KUKA KRL program: exampleKukaPath.src, exampleKukaPath.dat

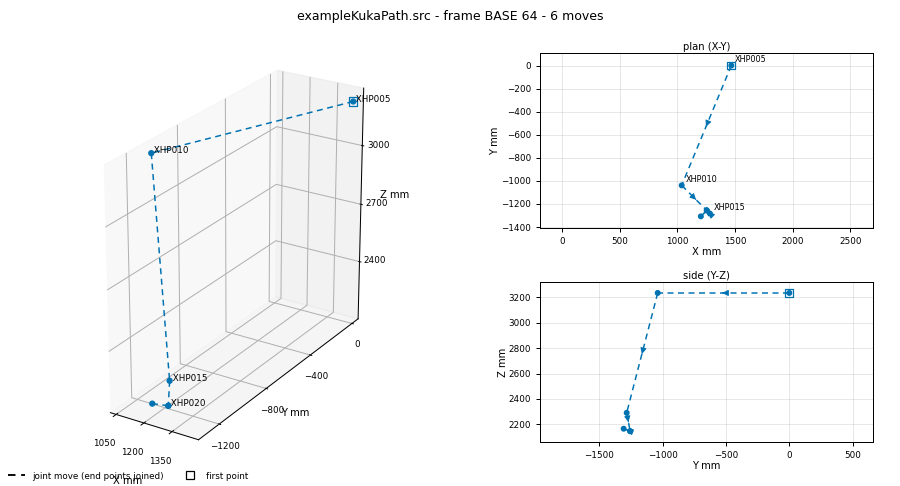
[picture p0: tool path of exampleKukaPath.src in frame BASE 64, 6 of 6 moves have a stored position in this frame; points joined in program order, loops and branches not executed]
--- exampleKukaPath.src ---
&ACCESS RVO1
&REL 274
&COMMENT Bld
&PARAM DISKPATH = KRC:\R1\Program\Production\223
DEF msn223v_030_01_030r2( )

DECL INT SRCDATA
DECL FLOAT SCRDATAFLOAT, ADRa
DECL INT DATAS13

;FOLD INI
  ;FOLD BASISTECH INI
    GLOBAL INTERRUPT DECL 3 WHEN $IN[1]==TRUE DO IR_STOPM ( )
    INTERRUPT ON 3
    BAS (#INITMOV,0 )
  ;ENDFOLD (BASISTECH INI)
  ;FOLD USER INI
    ;Make your modifications here
  ;ENDFOLD (USER INI)
;ENDFOLD (INI)

WAIT FOR  ( $IN[126] )
$OUT[125]=TRUE
$OUT[161]=FALSE

COLLSTOP( 15, 1 ) ;not Interrupt-Controlled
USE_CD_PARAMS(1)

;FOLD PTP HP005 CONT Vel=100 % PDATHH Tool[64]:NULL [64]:NULL ;%{PE}
;FOLD Parameters ;%{h}
;Params IlfProvider=kukaroboter.basistech.inlineforms.movement.old; Kuka.IsGlobalPoint=False; Kuka.PointName=HP005; Kuka.BlendingEnabled=True; Kuka.MoveDataPtpName=PDATHH; Kuka.VelocityPtp=100; Kuka.CurrentCDSetIndex=0; Kuka.MovementParameterFieldEnabled=True; IlfCommand=PTP
;ENDFOLD
$BWDSTART = FALSE
PDAT_ACT = PPDATHH
FDAT_ACT = FHP005
BAS(#PTP_PARAMS, 100.0)
SET_CD_PARAMS (0)
PTP XHP005 C_DIS C_DIS
;ENDFOLD

;FOLD PTP HP010 CONT Vel=100 % PDATHH Tool[64]:NULL Base[64]:NULL ;%{PE}
;FOLD Parameters ;%{h}
;Params IlfProvider=kukaroboter.basistech.inlineforms.movement.old; Kuka.IsGlobalPoint=False; Kuka.PointName=HP010; Kuka.BlendingEnabled=True; Kuka.MoveDataPtpName=PDATHH; Kuka.VelocityPtp=100; Kuka.CurrentCDSetIndex=0; Kuka.MovementParameterFieldEnabled=True; IlfCommand=PTP
;ENDFOLD
$BWDSTART = FALSE
PDAT_ACT = PPDATHH
FDAT_ACT = FHP010
BAS(#PTP_PARAMS, 100.0)
SET_CD_PARAMS (0)
PTP XHP010 C_Dis
;ENDFOLD
;FOLD PTP HP015 CONT Vel=100 % PDATHH Tool[64]:NULL Base[64]: ;%{PE}
;FOLD Parameters ;%{h}
;Params IlfProvider=kukaroboter.basistech.inlineforms.movement.old; Kuka.IsGlobalPoint=False; Kuka.PointName=HP015; Kuka.BlendingEnabled=True; Kuka.MoveDataPtpName=PDATHH; Kuka.VelocityPtp=100; Kuka.CurrentCDSetIndex=0; Kuka.MovementParameterFieldEnabled=True; IlfCommand=PTP
;ENDFOLD
$BWDSTART = FALSE
PDAT_ACT = PPDATHH
FDAT_ACT = FHP015
BAS(#PTP_PARAMS, 100.0)
SET_CD_PARAMS (0)
PTP XHP015 C_Dis
;ENDFOLD
;FOLD PTP HP020 CONT Vel=100 % PDATHH Tool[64]:NULL Base[64]: ;%{PE}
;FOLD Parameters ;%{h}
;Params IlfProvider=kukaroboter.basistech.inlineforms.movement.old; Kuka.IsGlobalPoint=False; Kuka.PointName=HP020; Kuka.BlendingEnabled=True; Kuka.MoveDataPtpName=PDATHH; Kuka.VelocityPtp=100; Kuka.CurrentCDSetIndex=0; Kuka.MovementParameterFieldEnabled=True; IlfCommand=PTP
;ENDFOLD
$BWDSTART = FALSE
PDAT_ACT = PPDATHH
FDAT_ACT = FHP020
BAS(#PTP_PARAMS, 100.0)
SET_CD_PARAMS (0)
PTP XHP020 C_Dis
;ENDFOLD
;FOLD PTP HP025 Vel=100 % PDATHH Tool[64]:NULL Base[64]: ;%{PE}
;FOLD Parameters ;%{h}
;Params IlfProvider=kukaroboter.basistech.inlineforms.movement.old; Kuka.IsGlobalPoint=False; Kuka.PointName=HP025; Kuka.BlendingEnabled=False; Kuka.MoveDataPtpName=PDATHH; Kuka.VelocityPtp=100; Kuka.CurrentCDSetIndex=0; Kuka.MovementParameterFieldEnabled=True; IlfCommand=PTP
;ENDFOLD
$BWDSTART = FALSE
PDAT_ACT = PPDATHH
FDAT_ACT = FHP025
BAS(#PTP_PARAMS, 100.0)
SET_CD_PARAMS (0)
PTP XHP025
;ENDFOLD
;FOLD PTP HP030 Vel=100 % PDATHH Tool[64]:NULL Base[64]: ;%{PE}
;FOLD Parameters ;%{h}
;Params IlfProvider=kukaroboter.basistech.inlineforms.movement.old; Kuka.IsGlobalPoint=False; Kuka.PointName=HP030; Kuka.BlendingEnabled=False; Kuka.MoveDataPtpName=PDATHH; Kuka.VelocityPtp=100; Kuka.CurrentCDSetIndex=0; Kuka.MovementParameterFieldEnabled=True; IlfCommand=PTP
;ENDFOLD
$BWDSTART = FALSE
PDAT_ACT = PPDATHH
FDAT_ACT = FHP030
BAS(#PTP_PARAMS, 100.0)
SET_CD_PARAMS (0)
PTP XHP030
;ENDFOLD

$OUT[125]=TRUE
$OUT[161]=TRUE
COLLSTOP( 15, 2+0 )
USE_CD_PARAMS( 0)

END

GLOBAL DEFFCT BOOL nearE6Pos(ePOS:IN)
 DECL E6POS ePOS

 DECL E6POS Delta
 DECL BOOL bRet

 bRet = False

 Delta.X = ABS(ePOS.X - $Pos_Act.X)
 Delta.Y = ABS(ePOS.Y - $Pos_Act.Y)
 Delta.Z = ABS(ePOS.Z - $Pos_Act.Z)
 Delta.A = ABS(ePOS.A - $Pos_Act.A)
 Delta.B = ABS(ePOS.B - $Pos_Act.B)
 Delta.C = ABS(ePOS.C - $Pos_Act.C)

 Delta.S = ePOS.S - $Pos_Act.S
 Delta.T = ePOS.T - $Pos_Act.T

 Delta.E1 = ABS(ePOS.E1 - $Pos_Act.E1)
 Delta.E2 = ABS(ePOS.E2 - $Pos_Act.E2)
 Delta.E3 = ABS(ePOS.E3 - $Pos_Act.E3)
 Delta.E4 = ABS(ePOS.E4 - $Pos_Act.E4)
 Delta.E5 = ABS(ePOS.E5 - $Pos_Act.E5)
 Delta.E6 = ABS(ePOS.E6 - $Pos_Act.E6)

 bRet= (Delta.X < MaxPosTol.X) and (Delta.Y < MaxPosTol.Y) and (Delta.Z < MaxPosTol.Z) and (Delta.A < MaxPosTol.A) and (Delta.B < MaxPosTol.B) and (Delta.C < MaxPosTol.C)
 bRet=bRet and (Delta.S == 0) and (Delta.T == 0)
 bRet=bRet and (Delta.E1 < MaxPosTol.E1) and (Delta.E2 < MaxPosTol.E2) and (Delta.E3 < MaxPosTol.E3) and (Delta.E4 < MaxPosTol.E4) and (Delta.E5 < MaxPosTol.E5) and (Delta.E6 < MaxPosTol.E6)
 Return(bRet)
ENDFCT

--- exampleKukaPath.dat ---
&ACCESS RVO1
&REL 274
&COMMENT Blindnietmutter setzen
&PARAM DISKPATH = KRC:\R1\Program\Production\223
DEFDAT  MSN223V_030_01_030R2
;FOLD EXTERNAL DECLARATIONS;%{PE}%MKUKATPBASIS,%CEXT,%VCOMMON,%P

;FOLD BASISTECH EXT;%{PE}%MKUKATPBASIS,%CEXT,%VEXT,%P
EXT  BAS (BAS_COMMAND  :IN,REAL  :IN )
DECL INT SUCCESS, FAIL, PROG
;ENDFOLD (BASISTECH EXT)

;FOLD USER EXT;%{E}%MKUKATPUSER,%CEXT,%VEXT,%P
;Make here your modifications
BOOL PROC_OK=FALSE

;FOLD COLLISION
EXT  COLLSTOP (INT  :IN,INT  :IN )
;ENDFOLD  (Collision)
;ENDFOLD (USER EXT)
;ENDFOLD (EXTERNAL DECLERATIONS)

DECL BOOL $BWDSTART = FALSE
DECL PDAT PDAT_ACT ={VEL 50.0000,ACC 50.0000,APO_DIST 100.000,APO_MODE #CDIS,GEAR_JERK 100.000,EXAX_IGN 0}
DECL FDAT FDAT_ACT = {TOOL_NO 64,BASE_NO 64,IPO_FRAME #BASE,POINT2[] " "}


; E6POS declarations
DECL E6POS XHP005={X 1468.736,Y 0.0,Z 3235.954,A 0.0,B 45.0,C 0.0,S 18,T 2,E1 0.0,E2 0.0,E3 0.0,E4 0.0,E5 0.0,E6 0.0}
DECL E6POS XHP010={X 1038.553,Y -1038.553,Z 3235.954,A -45.0,B 45.0,C 0.0,S 18,T 2,E1 0.0,E2 0.0,E3 0.0,E4 0.0,E5 0.0,E6 0.0}
DECL E6POS XHP015={X 1283.399,Y -1283.399,Z 2290.000,A 0.0,B 90.0,C 45.0,S 18,T 2,E1 0.0,E2 0.0,E3 0.0,E4 0.0,E5 0.0,E6 0.0}
DECL E6POS XHP020={X 1255.926,Y -1255.926,Z 2145.000,A -45.000,B 120.000,C 0.0,S 18,T 2,E1 0.0,E2 0.0,E3 0.0,E4 0.0,E5 0.0,E6 0.0}
DECL E6POS XHP025={X 1255.926,Y -1255.926,Z 2145.000,A 4.107,B 131.410,C 40.893,S 18,T 2,E1 0.0,E2 0.0,E3 0.0,E4 0.0,E5 0.0,E6 0.0}
DECL E6POS XHP030={X 1204.661,Y -1307.191,Z 2164.426,A 16.813,B 156.452,C 61.813,S 18,T 2,E1 0.0,E2 0.0,E3 0.0,E4 0.0,E5 0.0,E6 0.0}


; FDAT declarations
DECL FDAT FHP005={TOOL_NO 64,BASE_NO 64,IPO_FRAME #BASE,POINT2[] " "}
DECL FDAT FHP010={TOOL_NO 64,BASE_NO 64,IPO_FRAME #BASE,POINT2[] " "}
DECL FDAT FHP015={TOOL_NO 64,BASE_NO 64,IPO_FRAME #BASE,POINT2[] " "}
DECL FDAT FHP020={TOOL_NO 64,BASE_NO 64,IPO_FRAME #BASE,POINT2[] " "}
DECL FDAT FHP025={TOOL_NO 64,BASE_NO 64,IPO_FRAME #BASE,POINT2[] " "}
DECL FDAT FHP030={TOOL_NO 64,BASE_NO 64,IPO_FRAME #BASE,POINT2[] " "}


; LDAT declarations
DECL LDAT LLDATHH={VEL 0.200000,ACC 100.000,APO_DIST 500.000,APO_FAC 50.0000,AXIS_VEL 100.000,AXIS_ACC 100.000,ORI_TYP #VAR,CIRC_TYP #BASE,JERK_FAC 50.0000,GEAR_JERK 100.000,EXAX_IGN 0}
DECL LDAT LLDATHM={VEL 2.00000,ACC 100.000,APO_DIST 100.000,APO_FAC 50.0000,AXIS_VEL 100.000,AXIS_ACC 100.000,ORI_TYP #VAR,CIRC_TYP #BASE,JERK_FAC 50.0000,GEAR_JERK 100.000,EXAX_IGN 0}
DECL LDAT LLDATHL={VEL 2.00000,ACC 100.000,APO_DIST 30.0000,APO_FAC 50.0000,AXIS_VEL 100.000,AXIS_ACC 100.000,ORI_TYP #VAR,CIRC_TYP #BASE,JERK_FAC 50.0000,GEAR_JERK 100.000,EXAX_IGN 0}
DECL LDAT LLDATMH={VEL 2.00000,ACC 50.0000,APO_DIST 500.000,APO_FAC 50.0000,AXIS_VEL 100.000,AXIS_ACC 100.000,ORI_TYP #VAR,CIRC_TYP #BASE,JERK_FAC 50.0000,GEAR_JERK 100.000,EXAX_IGN 0}
DECL LDAT LLDATMM={VEL 2.00000,ACC 50.0000,APO_DIST 100.000,APO_FAC 50.0000,AXIS_VEL 100.000,AXIS_ACC 100.000,ORI_TYP #VAR,CIRC_TYP #BASE,JERK_FAC 50.0000,GEAR_JERK 100.000,EXAX_IGN 0}
DECL LDAT LLDATML={VEL 2.00000,ACC 50.0000,APO_DIST 30.0000,APO_FAC 50.0000,AXIS_VEL 100.000,AXIS_ACC 100.000,ORI_TYP #VAR,CIRC_TYP #BASE,JERK_FAC 50.0000,GEAR_JERK 100.000,EXAX_IGN 0}
DECL LDAT LLDATLH={VEL 2.00000,ACC 25.0000,APO_DIST 500.000,APO_FAC 50.0000,AXIS_VEL 100.000,AXIS_ACC 100.000,ORI_TYP #VAR,CIRC_TYP #BASE,JERK_FAC 50.0000,GEAR_JERK 100.000,EXAX_IGN 0}
DECL LDAT LLDATLM={VEL 2.00000,ACC 25.0000,APO_DIST 100.000,APO_FAC 50.0000,AXIS_VEL 100.000,AXIS_ACC 100.000,ORI_TYP #VAR,CIRC_TYP #BASE,JERK_FAC 50.0000,GEAR_JERK 100.000,EXAX_IGN 0}
DECL LDAT LLDATLL={VEL 2.00000,ACC 25.0000,APO_DIST 30.0000,APO_FAC 50.0000,AXIS_VEL 100.000,AXIS_ACC 100.000,ORI_TYP #VAR,CIRC_TYP #BASE,JERK_FAC 50.0000,GEAR_JERK 100.000,EXAX_IGN 0}

; PDAT declarations
DECL PDAT PPDATHH={VEL 50.0000,ACC 50.0000,APO_DIST 100.000,APO_MODE #CDIS,GEAR_JERK 100.000,EXAX_IGN 0}
DECL PDAT PPDATHM={VEL 100.000,ACC 100.000,APO_DIST 500.000,APO_MODE #CDIS,GEAR_JERK 100.000,EXAX_IGN 0}
DECL PDAT PPDATHL={VEL 100.000,ACC 100.000,APO_DIST 100.000,APO_MODE #CDIS,GEAR_JERK 100.000,EXAX_IGN 0}
DECL PDAT PPDATMH={VEL 100.000,ACC 50.0000,APO_DIST 1000.00,APO_MODE #CDIS,GEAR_JERK 100.000,EXAX_IGN 0}
DECL PDAT PPDATMM={VEL 100.000,ACC 50.0000,APO_DIST 500.000,APO_MODE #CDIS,GEAR_JERK 100.000,EXAX_IGN 0}
DECL PDAT PPDATML={VEL 100.000,ACC 50.0000,APO_DIST 100.000,APO_MODE #CDIS,GEAR_JERK 100.000,EXAX_IGN 0}
DECL PDAT PPDATLH={VEL 100.000,ACC 25.0000,APO_DIST 1000.00,APO_MODE #CDIS,GEAR_JERK 100.000,EXAX_IGN 0}
DECL PDAT PPDATLM={VEL 100.000,ACC 25.0000,APO_DIST 500.000,APO_MODE #CDIS,GEAR_JERK 100.000,EXAX_IGN 0}
DECL PDAT PPDATLL={VEL 100.000,ACC 25.0000,APO_DIST 100.000,APO_MODE #CDIS,GEAR_JERK 100.000,EXAX_IGN 0}

DECL MODULEPARAM_T LAST_TP_PARAMS={PARAMS[] "Kuka.PointName=HP115; Kuka.FrameData.base_no=1; Kuka.FrameData.tool_no=1; Kuka.FrameData.ipo_frame=#BASE; Kuka.FrameData.point2=; Kuka.isglobalpoint=False; Kuka.MoveDataPtpName=PDATHH; Kuka.MovementDataPdat.apo_mode=#CDIS; Kuka.MovementDataPdat.apo_dist=100; Kuka.MovementData.vel=50; Kuka.MovementData.acc=50; Kuka.MovementData.gear_jerk=100; Kuka.MovementData.exax_ign=0; Kuka.VelocityPtp=50; Kuka.BlendingEnabled=False; Kuka.CurrentCDSetIndex=0; Kuka.MoveDataName=LDATHH; Kuka.MovementData.apo_fac=50; Kuka.MovementData.apo_dist=500; Kuka.MovementData.axis_acc=100; Kuka.MovementData.axis_vel=100; Kuka.MovementData.circ_typ=#BASE; Kuka.MovementData.jerk_fac=50; Kuka.MovementData.ori_typ=#VAR; Kuka.VelocityPath=0.2                                                                                                                     "}

ENDDAT
